(* CODESYS project fscontrollertoolbox_0.1.0.library
   Company: FisoThemes
   DocFormat: reStructuredText
   Description: A library for building and modelling control systems.
   Version: 0.1.0
   Placeholder: FsControllerToolbox
   Author: Goodwill Mzumala
   Title: FsControllerToolbox

Project tree, tasks and I/O mapping:
  libraries: FsCommon, * (FisoThemes); Tc2_Standard, * (Beckhoff Automation GmbH); Tc2_System, * (Beckhoff Automation GmbH); Tc3_Module, * (Beckhoff Automation GmbH); Tc2_Math, * (Beckhoff Automation GmbH)
  Analysis/
  Conditioning/
    DUTs/
      data type E_DeadbandMode
    function block FB_Deadband [ST]: FB_init, Maximum, Minimum, Mode, Reset, Run
    function block FB_Hysteresis [ST]: FB_init, LowerThreshold, Output, Reset, Run, UpperThreshold
  Control/
    DUTs/
      data type E_AntiWindupMethod
    function block FB_Differentiator [ST]: FB_init, Reset, Run, Td, Tv
    function block FB_Integrator [ST]: AntiWindupActive, AntiWindupMethod, FB_init, Maximum, Minimum, Reset, Run, Sync, Tn, TrackingTimeConstant
    function block FB_ProportionalGain [ST]: FB_init, Kp, Reset, Run
  Filter/
    function block FB_FirstOrderIIRFilter [ST]: Alpha, FB_init, Reset, Run
  Internal/
    program PLAYGROUND [ST]
  Project Information/
    function F_GetCompany [ST]
    function F_GetTitle [ST]
    function F_GetVersion [ST]
  Shared/
    ITFs/
      interface I_Component
      interface I_Resettable: Reset
      interface I_SiComponent: Input
      interface I_SisoComponent: Input, Output
      interface I_SoComponent: Output
    function block FB_SiComponent [ST]: Input
    function block FB_SisoComponent [ST]: Input, Output
    function block FB_SoComponent [ST]: Output
  Signals/
    DUTs/
      data type E_RampDirection
    ITFs/
      interface I_PeriodicSignal: Amplitude, Bias, Period, Phase
    function block FB_PeriodicSignal [ST]: Amplitude, Bias, Period, Phase
    function block FB_PWM [ST]: DutyCycle, FB_init, IsHigh, Reset, Run
    function block FB_Ramp [ST]: FB_init, Rate, Reset, Run, StartValue
    function block FB_SawtoothWave [ST]: Direction, FB_init, Reset, Run
    function block FB_SineWave [ST]: FB_init, Reset, Run
    function block FB_SquareWave [ST]: FB_init, Reset, Run
    function block FB_TriangleWave [ST]: FB_init, Reset, Run
  Simulation/
    function block FB_FirstOrderPlant [ST]: FB_init, Gain, Reset, Run, Tau
    function block FB_SecondOrderPlant [ST]: FB_init, Gain, Reset, Run, Wn, Zeta
  Transform/
  Version/
    global variables Global_Version
*)

// Conditioning/DUTs/E_DeadbandMode
(*
Specifies the behaviour of :itf:`FB_Deadband` when the input is within the band.
*)
{attribute 'qualified_only'}
{attribute 'strict'}
{attrubute 'to_string'}
TYPE E_DeadbandMode :
(
	Hold := 0, // Output holds its last value while the input is within the band.
	Zero := 1  // Output is set to zero while the input is within the band.
)BYTE;
END_TYPE

// Control/DUTs/E_AntiWindupMethod
(*
Specifies the anti-windup strategy used by :itf:`FB_Integrator`.
*)
{attribute 'qualified_only'}
{attribute 'strict'}
{attribute 'to_string'}
TYPE E_AntiWindupMethod :
(
	// Halts integration when the output is saturated.
	Clamping        := 0, 
	// Feeds back the saturation error to unwind the integrator gradually. 
	// Recommended for slow systems with significant lag
	BackCalculation := 1
)BYTE;
END_TYPE

// Signals/DUTs/E_RampDirection
(* Specifies the direction of a ramping signal. *)
{attribute 'qualified_only'}
{attribute 'strict'}
{attribute 'to_string'}
TYPE E_RampDirection :
(
	Rising   := 0, // Output increases over time.
	Falling  := 1  // Output decreases over time.
)BYTE;
END_TYPE

// Version/Global_Version
{attribute 'TcGenerated'}
{attribute 'no-analysis'}
{attribute 'linkalways'}
// This function has been automatically generated from the project information.
VAR_GLOBAL CONSTANT
	{attribute 'const_non_replaced'}
	stLibVersion_FsControllerToolbox : ST_LibVersion := (iMajor := 0, iMinor := 1, iBuild := 0, iRevision := 0, nFlags := 0, sVersion := '0.1.0');
END_VAR

// Conditioning/FB_Deadband
(*
Suppresses small input signals within a configurable band.

When the input falls within [:attr:`Minimum`, :attr:`Maximum`], the output
is either zeroed or held at its last value depending on :attr:`Mode`. Outside
the band the input passes through unchanged.

.. note::
   The block is ``FINAL`` and must be instantiated, not extended.
   Use ``FB_init`` to set :attr:`fMinimum`, :attr:`fMaximum`, and :attr:`eMode`
   at declaration time.
*)
{attribute 'no_assign'}
{attribute 'enable_dynamic_creation'}
{attribute 'no_explicit_call' := 'direct call for this function block is not allowed'}
FUNCTION_BLOCK FINAL FB_Deadband EXTENDS FB_SisoComponent
IMPLEMENTS FsCommon.I_Runnable, I_Resettable
VAR
	_fMinimum : LREAL; // Lower bound of the deadband. Clamped to <= Maximum.
	_fMaximum : LREAL; // Upper bound of the deadband. Clamped to >= Minimum.
	_eMode    : E_DeadbandMode; // Output behaviour when input is within the band.
END_VAR

METHOD FB_init : BOOL
VAR_INPUT
	bInitRetains : BOOL;  // if TRUE, the retain variables are initialized (warm start / cold start)
	bInCopyCode  : BOOL;  // if TRUE, the instance afterwards gets moved into the copy code (online change)
	fMaximum     : LREAL; // Upper bound of the deadband.
	fMinimum     : LREAL; // Lower bound of the deadband.
	eMode        : E_DeadbandMode; // Output behaviour when the input is within the band.
END_VAR
THIS^.Maximum  := fMaximum;
THIS^.Minimum  := fMinimum;
THIS^._eMode   := eMode;
END_METHOD

(*
Gets or sets the upper bound of the deadband.

Internally clamped to be greater than or equal to :attr:`Minimum`.
Set this before :attr:`Minimum` to ensure the guard applies correctly.
*)
PROPERTY Maximum : LREAL
GET
Maximum := THIS^._fMaximum;
END_GET
SET
THIS^._fMaximum := MAX(THIS^._fMinimum, Maximum);
END_SET
END_PROPERTY

(*
Gets or sets the lower bound of the deadband.

Internally clamped to be less than or equal to :attr:`Maximum`.
Set :attr:`Maximum` before this property to ensure the guard applies correctly.
*)
PROPERTY Minimum : LREAL
GET
Minimum := THIS^._fMinimum;
END_GET
SET
THIS^._fMinimum := MIN(THIS^._fMaximum, Minimum);
END_SET
END_PROPERTY

(*
Gets or sets the output behaviour when the input is within the band.

:attr:`~E_DeadbandMode.Zero` sets the output to zero. 
:attr:`~E_DeadbandMode.Hold` retains the last output value. 

Changes take effect on th next :meth:`Run` call.
*)
PROPERTY Mode : E_DeadbandMode
GET
Mode := THIS^._eMode;
END_GET
SET
THIS^._eMode := Mode;
END_SET
END_PROPERTY

(* 
Resets the output to a value consistent with the current mode. 

In :attr:`~E_DeadbandMode.Zero` mode the output is set to zero.
In :attr:`~E_DeadbandMode.Hold` mode the output is set to the current input.
*)
METHOD Reset
VAR_INPUT
END_VAR
CASE THIS^._eMode OF
	E_DeadbandMode.Hold:
		THIS^._fOutput := THIS^._fInput;
	E_DeadbandMode.Zero:
		THIS^._fOutput := 0;
END_CASE
END_METHOD

(* Applies the deadband to the current input. *)
METHOD Run
VAR_INPUT
END_VAR
THIS^._fMaximum := MAX(THIS^._fMinimum, THIS^._fMaximum);
THIS^._fMinimum := MIN(THIS^._fMinimum, THIS^._fMaximum);

IF THIS^._fInput >= THIS^._fMinimum AND THIS^._fInput <= THIS^._fMaximum THEN
    CASE THIS^._eMode OF
        E_DeadbandMode.Zero:
            THIS^._fOutput := 0;
        E_DeadbandMode.Hold:
            ; // Output retains its last value.
    END_CASE
ELSE
    THIS^._fOutput := THIS^._fInput;
END_IF
END_METHOD

END_FUNCTION_BLOCK

// Shared/FB_SisoComponent
(*
Abstract function block providing :attr:`Input` and :attr:`Output` properties
for single-input single-output controller toolbox components.

.. NOTE::
   Direct calls to this function block are not permitted (``no_explicit_call``).
*)
{attribute 'no_explicit_call' := 'direct call for this function block is not allowed'}
FUNCTION_BLOCK ABSTRACT FB_SisoComponent
IMPLEMENTS I_SisoComponent, I_SiComponent, I_SoComponent
VAR
	_fInput 	: LREAL;
	_fOutput 	: LREAL;
END_VAR

(* Gets or sets the input to the component.*)
PROPERTY Input : LREAL
GET
Input := THIS^._fInput;
END_GET
SET
THIS^._fInput := Input;
END_SET
END_PROPERTY

(* Gets the output produced by the component.*)
PROPERTY Output : LREAL
GET
Output := THIS^._fOutput;
END_GET
END_PROPERTY

END_FUNCTION_BLOCK

// Shared/ITFs/I_SisoComponent
(*
Interface for single-input single-output controller toolbox components.

Implementors expose a writable :attr:`Input` and a read-only :attr:`Output`,
both as ``LREAL``.
*)
INTERFACE I_SisoComponent EXTENDS I_Component

// Gets or sets the input to the component.
PROPERTY Input : LREAL
GET
END_GET
SET
END_SET
END_PROPERTY

// Gets the output produced by the component.
PROPERTY Output : LREAL
GET
END_GET
END_PROPERTY

END_INTERFACE

// Shared/ITFs/I_Component
(*
Base interface for all FsControllerToolbox components.

Extends ``__SYSTEM.IQueryInterface`` to allow runtime type checking via
``__QUERYINTERFACE``.
*)
INTERFACE I_Component EXTENDS __SYSTEM.IQueryInterface

END_INTERFACE

// Shared/ITFs/I_SiComponent
(*
Interface for single-input controller toolbox components.

Implementors expose a write-only :attr:`Input` property. For components that
also produce an output signal, use :itf:`I_SisoComponent` instead.
*)
INTERFACE I_SiComponent

// Gets or sets the input to the component.
PROPERTY Input : LREAL
GET
END_GET
SET
END_SET
END_PROPERTY

END_INTERFACE

// Shared/ITFs/I_SoComponent
(*
Interface for single-output controller toolbox components.

Implementors expose a read-only :attr:`Output` property. For components that
also accept an input signal, use :itf:`I_SisoComponent` instead.
*)
INTERFACE I_SoComponent EXTENDS I_Component

// Gets the output produced by the component.
PROPERTY Output : LREAL
GET
END_GET
END_PROPERTY

END_INTERFACE

// Shared/ITFs/I_Resettable
(*
Interface for components that can be returned to a known initial state.

Implementors must define :meth:`Reset` to clear any internal state, such as
accumulators, filter history, or elapsed time, and restore the output to its
initial condition.
*)
INTERFACE I_Resettable EXTENDS __SYSTEM.IQueryInterface

(* Clears internal state and restores the component to its initial condition. *)
METHOD Reset
VAR_INPUT
END_VAR
END_METHOD

END_INTERFACE

// Conditioning/FB_Hysteresis
(*
Implements a hysteresis controller with two thresholds and latching behaviour.

The output switches low when the input rises above :attr:`UpperThreshold` and
switches high when the input falls below :attr:`LowerThreshold`. Between the
two thresholds the output latches at its current state.

This convention suits heating applications, the output drives a heater that
turns on when the process falls below the lower threshold and off when it
exceeds the upper threshold.

.. note::
   The block is ``FINAL`` and must be instantiated, not extended.
   Use ``FB_init`` to set :attr:`fUpperThreshold` and :attr:`fLowerThreshold`
   at declaration time.
*)
{attribute 'no_assign'}
{attribute 'enable_dynamic_creation'}
{attribute 'no_explicit_call' := 'direct call for this function block is not allowed'}
FUNCTION_BLOCK FINAL FB_Hysteresis EXTENDS FB_SiComponent
IMPLEMENTS FsCommon.I_Runnable, I_Resettable
VAR
	_fUpperThreshold : LREAL; // Input level above which the output switches low.
	_fLowerThreshold : LREAL; // Input level below which the output switches high.
	_bOutput         : BOOL;  // Current output state.
END_VAR

METHOD FB_init : BOOL
VAR_INPUT
	bInitRetains 	 : BOOL; // if TRUE, the retain variables are initialized (warm start / cold start)
	bInCopyCode 	 : BOOL;  // if TRUE, the instance afterwards gets moved into the copy code (online change)
	fUpperThreshold  : LREAL; // Input level above which the output switches low.
	fLowerThreshold  : LREAL; // Input level below which the output switches high.
END_VAR
THIS^._fUpperThreshold := fUpperThreshold;
THIS^._fLowerThreshold := fLowerThreshold;
END_METHOD

(*
Gets or sets the lower threshold.

When the input falls below this value the output switches high. Must be less
than :attr:`UpperThreshold` for correct operation.
*)
PROPERTY LowerThreshold : LREAL
GET
LowerThreshold := THIS^._fLowerThreshold;
END_GET
SET
THIS^._fLowerThreshold := LowerThreshold;
END_SET
END_PROPERTY

(*
Gets the current output state. 

TRUE when the process is below :attr:`LowerThreshold`.
FALSE when above :attr:`UpperThreshold`.
*)
PROPERTY Output : BOOL
GET
Output := THIS^._bOutput;
END_GET
END_PROPERTY

(*
Evaluates the current input against the thresholds and sets the output immediately,
rather than waiting for the input to cross a threshold.

If the input is above :attr:`UpperThreshold` the output is set low. If below
:attr:`LowerThreshold` the output is set high. If between the two thresholds
the output defaults to low as a safe state.
*)
METHOD Reset
VAR_INPUT
END_VAR
THIS^._bOutput := THIS^._fInput < THIS^._fLowerThreshold;
END_METHOD

(* Evaluates the input against the thresholds and updates the output. *)
METHOD Run
VAR_INPUT
END_VAR
IF THIS^._fInput > THIS^._fUpperThreshold THEN
	THIS^._bOutput := FALSE;
ELSIF THIS^._fInput < THIS^._fLowerThreshold THEN
	THIS^._bOutput := TRUE;
END_IF
END_METHOD

(*
Gets or sets the upper threshold.

When the input rises above this value the output switches low. Must be greater
than :attr:`LowerThreshold` for correct operation.
*)
PROPERTY UpperThreshold : LREAL
GET
UpperThreshold := THIS^._fUpperThreshold;
END_GET
SET
THIS^._fUpperThreshold := UpperThreshold;
END_SET
END_PROPERTY

END_FUNCTION_BLOCK

// Shared/FB_SiComponent
(*
Abstract function block providing an :attr:`Input` property for single-input
controller toolbox components.

Concrete implementations read from ``_fInput`` to consume the signal written
by the caller.

.. note::
   Direct calls to this function block are not permitted (``no_explicit_call``).
   Extend it and call the derived block instead.
*)
{attribute 'no_explicit_call' := 'direct call for this function block is not allowed'}
FUNCTION_BLOCK ABSTRACT FB_SiComponent
IMPLEMENTS I_SiComponent
VAR
    _fInput : LREAL;
END_VAR

(* Gets or sets the input to the component.*)
PROPERTY Input : LREAL
GET
Input := THIS^._fInput;
END_GET
SET
THIS^._fInput := Input;
END_SET
END_PROPERTY

END_FUNCTION_BLOCK

// Control/FB_Differentiator
(*
Differentiates the input signal with an optional first-order damping filter.

The transfer function is:

.. math::

   D(s) = \frac{T_v \cdot s}{T_d \cdot s + 1}

where :math:`T_v` is :attr:`Tv` and :math:`T_d` is :attr:`Td`. The filter is
discretised using the Tustin (bilinear) method.

Setting :attr:`Tv` to ``LTIME#0`` disables the derivative term entirely.
Setting :attr:`Td` to ``LTIME#0`` removes the damping filter, giving a pure
derivative. This is not recommended in practice due to noise sensitivity.

.. note::
   If derivative kick on setpoint steps is undesirable, pass the negated
   process variable as :attr:`Input` rather than the full error. The integrator
   should still receive the full error signal.

   The block is ``FINAL`` and must be instantiated, not extended.
   Use ``FB_init`` to set :attr:`tTv` and :attr:`tTd` at declaration time.
*)
{attribute 'no_assign'}
{attribute 'enable_dynamic_creation'}
{attribute 'no_explicit_call' := 'direct call for this function block is not allowed'}
FUNCTION_BLOCK FINAL FB_Differentiator EXTENDS FB_SisoComponent
IMPLEMENTS FsCommon.I_Runnable, I_Resettable
VAR
	_tTv          : LTIME; // Rate time (Tv). Determines derivative action strength.
	_tTd          : LTIME; // Damping time (Td). Filters the derivative signal to reduce noise sensitivity.
	_fPrevInput   : LREAL; // Input from the previous cycle.
	_fFilterState : LREAL; // Internal state of the damping filter.
END_VAR

METHOD FB_init : BOOL
VAR_INPUT
	bInitRetains : BOOL; // if TRUE, the retain variables are initialized (warm start / cold start)
	bInCopyCode  : BOOL;  // if TRUE, the instance afterwards gets moved into the copy code (online change)
	tTv          : LTIME; // Rate time. T#0S disables the derivative term entirely.
	tTd          : LTIME; // Damping time. LTIME#0 means no filtering (pure derivative).
END_VAR
THIS^._tTv := tTv;
THIS^._tTd := tTd;
END_METHOD

(*
Clears the filter state and output. 
Sets the previous input to the current input to avoid a spike on the next :meth:`Run` call. 
*)
METHOD Reset
VAR_INPUT
END_VAR
THIS^._fFilterState := 0;
THIS^._fPrevInput   := THIS^._fInput;
THIS^._fOutput      := 0;
END_METHOD

(*
Advances the differentiator by one time step.

On the first call the cycle time is measured, the filter state is initialised,
and the method returns early without producing an output. This prevents a spike
caused by an uninitialised previous input.

.. note::
   Must be called once per cycle on a single PLC task. If :attr:`Tv` is
   ``LTIME#0`` the output is held at zero.
*)
METHOD Run
VAR_INST
	{attribute 'hide'}
	bInit       : BOOL := TRUE;
	{attribute 'hide'}
	fT          : LREAL;
	{attribute 'hide'}
	fbTaskCycle : FsCommon.FB_PlcTaskCycleChangeDetector(0);
END_VAR
VAR
	fTv            : LREAL;
	fTd            : LREAL;
	fDen           : LREAL;
	fAlpha         : LREAL;
	fRawDerivative : LREAL;
END_VAR
IF bInit THEN
	fT := TO_LREAL(FsCommon.F_GetCurrentTaskCycleTime()) / TO_LREAL(LTIME#1S);
	RETURN(bInit := fT <= 0);
	fbTaskCycle.TaskIndex := FsCommon.F_GetCurrentTaskIndex();
	THIS^._fPrevInput     := THIS^._fInput;
	THIS^._fFilterState   := 0;
	RETURN;
END_IF

RETURN(NOT fbTaskCycle.HasChanged);

IF THIS^._tTv = LTIME#0S THEN
	THIS^._fOutput    := 0;
	THIS^._fPrevInput := THIS^._fInput;
	RETURN;
END_IF

fTv := TO_LREAL(THIS^._tTv) / TO_LREAL(LTIME#1S);
fTd := TO_LREAL(THIS^._tTd) / TO_LREAL(LTIME#1S);

fRawDerivative := fTv * (THIS^._fInput - THIS^._fPrevInput) / fT;

IF THIS^._tTd = LTIME#0S THEN
	THIS^._fOutput := fRawDerivative;
ELSE
	fDen                := fTd + fT / 2.0;
	fAlpha              := (fTd - fT / 2.0) / fDen;
	THIS^._fFilterState := fAlpha * THIS^._fFilterState + (1.0 - fAlpha) * fRawDerivative;
	THIS^._fOutput      := THIS^._fFilterState;
END_IF

THIS^._fPrevInput := THIS^._fInput;
END_METHOD

(*
Gets or sets the damping time (Td).

This filters the derivative signal to reduce sensitivity to noise. A longer
value gives more filtering but reduces derivative effectiveness. Setting it
to ``LTIME#0`` removes the filter entirely, giving a pure derivative (not
recommended in practice due to noise sensitivity).
*)
PROPERTY Td : LTIME
GET
Td := THIS^._tTd;
END_GET
SET
THIS^._tTd := Td;
END_SET
END_PROPERTY

(*
Gets or sets the rate time (Tv).

This controls how strongly the block reacts to changes in the input. A longer
value increases derivative action. Setting it to ``LTIME#0`` disables the
derivative term entirely, holding the output at zero.
*)
PROPERTY Tv : LTIME
GET
Tv := THIS^._tTv;
END_GET
SET
THIS^._tTv := Tv;
END_SET
END_PROPERTY

END_FUNCTION_BLOCK

// Control/FB_Integrator
(*
Integrates the input error signal over time.

The output accumulates the input scaled by the integral gain :math:`K_i = 1 / T_n`,
and is clamped to [:attr:`Minimum`, :attr:`Maximum`] on every cycle. Two anti-windup
strategies are available via :attr:`AntiWindupMethod`.

Setting :attr:`Tn` to ``LTIME#0`` disables integration, holding the output at
its current integrator state.

.. note::
   Set :attr:`Maximum` before :attr:`Minimum` to ensure the clamp is applied
   correctly. Setting :attr:`Minimum` first may cause it to be clamped against
   an uninitialised :attr:`Maximum`.

   The block is ``FINAL`` and must be instantiated, not extended.
   Use ``FB_init`` to set :attr:`tTn`, :attr:`fMaximum`, :attr:`fMinimum`,
   :attr:`eAntiWindupMethod`, and :attr:`tTrackingTimeConstant` at declaration time.
*)
{attribute 'no_assign'}
{attribute 'enable_dynamic_creation'}
{attribute 'no_explicit_call' := 'direct call for this function block is not allowed'}
FUNCTION_BLOCK FINAL FB_Integrator EXTENDS FB_SisoComponent
IMPLEMENTS FsCommon.I_Runnable, I_Resettable
VAR
	_tTn                   : LTIME; // Integral action time (Tn).
	_fMaximum              : LREAL :=  FsCommon.GVL_TypeValueLimits.LREAL_MAX; // Upper output clamp.
	_fMinimum              : LREAL :=  FsCommon.GVL_TypeValueLimits.LREAL_MIN; // Lower output clamp.
	_eAntiWindupMethod     : E_AntiWindupMethod; // Anti-windup strategy.
	_tTrackingTimeConstant : LTIME; // Tracking time constant (Tt) for back-calculation anti-windup.
	_fIntegratorState      : LREAL; // Internal integrator accumulator.
	_bAntiWindupActive     : BOOL;  // TRUE when the output is saturated and anti-windup is limiting integration.
	_bSync                 : BOOL;  // Triggers a bumpless transfer on the next Run call.
	_fSync                 : LREAL; // Target integrator state for bumpless transfer.
END_VAR

(* Gets whether the output is currently saturated and anti-windup is actively limiting integration. *)
PROPERTY AntiWindupActive : BOOL
GET
AntiWindupActive := THIS^._bAntiWindupActive;
END_GET
END_PROPERTY

(*
Gets or sets the anti-windup strategy.

:attr:`~E_AntiWindupMethod.Clamping` halts integration when the output is
saturated. :attr:`~E_AntiWindupMethod.BackCalculation` feeds the saturation
error back into the integrator gradually, which is better suited to slow
systems with significant lag such as thermal processes.
*)
PROPERTY AntiWindupMethod : E_AntiWindupMethod
GET
AntiWindupMethod := THIS^._eAntiWindupMethod;
END_GET
SET
THIS^._eAntiWindupMethod := AntiWindupMethod;
END_SET
END_PROPERTY

METHOD FB_init : BOOL
VAR_INPUT
	bInitRetains 		  : BOOL;  // if TRUE, the retain variables are initialized (warm start / cold start)
	bInCopyCode 		  : BOOL;  // if TRUE, the instance afterwards gets moved into the copy code (online change)
	tTn                   : LTIME; // Integral action time. LTIME#0 disables integration.
	fMaximum              : LREAL; // Upper output clamp.
	fMinimum              : LREAL; // Lower output clamp.
	eAntiWindupMethod     : E_AntiWindupMethod; // Anti-windup strategy.
	tTrackingTimeConstant : LTIME; // Tracking time constant for back-calculation anti-windup.
END_VAR
THIS^._tTn                   := tTn;
THIS^.Maximum                := fMaximum;
THIS^.Minimum                := fMinimum;
THIS^._eAntiWindupMethod     := eAntiWindupMethod;
THIS^._tTrackingTimeConstant := tTrackingTimeConstant;
END_METHOD

(*
Gets or sets the upper output clamp.

The output is clamped to this value on every cycle. Internally clamped to be
greater than or equal to :attr:`Minimum`. Set this before :attr:`Minimum` to
ensure the guard applies correctly.
*)
PROPERTY Maximum : LREAL
GET
Maximum := THIS^._fMaximum;
END_GET
SET
THIS^._fMaximum := MAX(THIS^._fMinimum, Maximum);
END_SET
END_PROPERTY

(*
Gets or sets the lower output clamp.

The output is clamped to this value on every cycle. Internally clamped to be
less than or equal to :attr:`Maximum`. Set :attr:`Maximum` before this property
to ensure the guard applies correctly.
*)
PROPERTY Minimum : LREAL
GET
Minimum := THIS^._fMinimum;
END_GET
SET
THIS^._fMinimum := MIN(THIS^._fMaximum, Minimum);
END_SET
END_PROPERTY

(* Clears the integrator state, output, and anti-windup flag. *)
METHOD Reset
VAR_INPUT
END_VAR
THIS^._fIntegratorState  := 0;
THIS^._fOutput           := 0;
THIS^._bAntiWindupActive := FALSE;
END_METHOD

(*
Advances the integrator by one time step.

.. note::
   Must be called once per cycle on a single PLC task. If :attr:`Tn` is
   ``LTIME#0`` the output is held at the current integrator state without
   further integration.
*)
METHOD Run
VAR_INST
	{attribute 'hide'}
	bInit       : BOOL := TRUE;
	{attribute 'hide'}
	fT          : LREAL;
	{attribute 'hide'}
	fbTaskCycle : FsCommon.FB_PlcTaskCycleChangeDetector(0);
END_VAR
VAR
	fKi                   : LREAL;
	fTt                   : LREAL;
	fWindupBack           : LREAL;
	fUnsat                : LREAL;
	fSaturated            : LREAL;
END_VAR
IF bInit THEN
	fT := TO_LREAL(FsCommon.F_GetCurrentTaskCycleTime()) / TO_LREAL(LTIME#1S);
	RETURN(bInit := fT <= 0);
	fbTaskCycle.TaskIndex := FsCommon.F_GetCurrentTaskIndex();
END_IF

THIS^._fMaximum := MAX(THIS^._fMinimum, THIS^._fMaximum);
THIS^._fMinimum := MIN(THIS^._fMinimum, THIS^._fMaximum);

RETURN(NOT fbTaskCycle.HasChanged);

// Bumpless transfer, force integrator state before anything else.
IF FsCommon.F_ResetOnTrue(THIS^._bSync) THEN
	THIS^._fIntegratorState := LIMIT(THIS^._fMinimum, THIS^._fSync, THIS^._fMaximum);
END_IF

IF THIS^._tTn = LTIME#0S THEN
	THIS^._fOutput := THIS^._fIntegratorState;
	RETURN;
END_IF

fKi := 1.0 / (TO_LREAL(THIS^._tTn) / TO_LREAL(LTIME#1S));

CASE THIS^._eAntiWindupMethod OF
	E_AntiWindupMethod.Clamping:
		IF NOT THIS^._bAntiWindupActive OR
		   (THIS^._fOutput >= THIS^._fMaximum AND THIS^._fInput < 0) OR
		   (THIS^._fOutput <= THIS^._fMinimum AND THIS^._fInput > 0) THEN
			THIS^._fIntegratorState :=
				THIS^._fIntegratorState + fKi * THIS^._fInput * fT;
		END_IF

	E_AntiWindupMethod.BackCalculation:
		fTt := TO_LREAL(THIS^._tTrackingTimeConstant) / TO_LREAL(LTIME#1S);
		fWindupBack := SEL(
			fTt > 0,
			0.0,
			(THIS^._fOutput - THIS^._fIntegratorState) / fTt);
		THIS^._fIntegratorState :=
			THIS^._fIntegratorState + (fKi * THIS^._fInput + fWindupBack) * fT;
END_CASE

fUnsat                   := THIS^._fIntegratorState;
fSaturated               := LIMIT(THIS^._fMinimum, fUnsat, THIS^._fMaximum);
THIS^._bAntiWindupActive := fSaturated <> fUnsat;
THIS^._fOutput           := fSaturated;
END_METHOD

(*
Forces the integrator state to a given value on the next :meth:`Run` call.

The value is clamped to [:attr:`Minimum`, :attr:`Maximum`] before being applied.
Use this for bumpless transfer when switching from manual to automatic mode,
to prevent a sudden jump in output.
*)
METHOD Sync
VAR_INPUT
	// Target integrator state.
	fValue : LREAL; 
END_VAR
THIS^._bSync := TRUE;
THIS^._fSync := LIMIT(THIS^._fMinimum, fValue, THIS^._fMaximum);
END_METHOD

(*
Gets or sets the integral action time (Tn).

This controls how aggressively the integrator responds to sustained error.
A shorter value increases integral action. Setting it to ``LTIME#0`` disables
integration entirely, holding the output at the current integrator state.
*)
PROPERTY Tn : LTIME
GET
Tn := THIS^._tTn;
END_GET
SET
THIS^._tTn := Tn;
END_SET
END_PROPERTY

(*
Gets or sets the tracking time constant (Tt) for back-calculation anti-windup.

This controls how quickly the integrator unwinds after saturation. A typical
starting value is ``SQRT(Tn * Td)``. Setting it to ``LTIME#0`` disables the
back-calculation correction. Ignored when :attr:`AntiWindupMethod` is
:attr:`~E_AntiWindupMethod.Clamping`.
*)
PROPERTY TrackingTimeConstant : LTIME
GET
TrackingTimeConstant := THIS^._tTrackingTimeConstant;
END_GET
SET
THIS^._tTrackingTimeConstant := TrackingTimeConstant;
END_SET
END_PROPERTY

END_FUNCTION_BLOCK

// Control/FB_ProportionalGain
(*
Applies a proportional gain to the input error signal.

The output is computed as:

.. math::

   y = K_p \cdot e

where :math:`K_p` is :attr:`Kp` and :math:`e` is the error signal set via :attr:`Input`.

.. note::
   The block is ``FINAL`` and must be instantiated, not extended.
   Use ``FB_init`` to set :attr:`fKp` at declaration time.
*)
{attribute 'no_assign'}
{attribute 'enable_dynamic_creation'}
{attribute 'no_explicit_call' := 'direct call for this function block is not allowed'}
FUNCTION_BLOCK FINAL FB_ProportionalGain EXTENDS FB_SisoComponent
IMPLEMENTS FsCommon.I_Runnable, I_Resettable
VAR
	_fKp : LREAL; // Proportional gain.
END_VAR

METHOD FB_init : BOOL
VAR_INPUT
	bInitRetains : BOOL; // if TRUE, the retain variables are initialized (warm start / cold start)
	bInCopyCode  : BOOL;  // if TRUE, the instance afterwards gets moved into the copy code (online change)
	fKp          : LREAL; // Proportional gain.
END_VAR
THIS^._fKp := fKp;
END_METHOD

(*
Gets or sets the proportional gain.

A higher value produces a stronger response to error but may cause overshoot.
A lower value produces a more gradual response. A value of 0 disables the
proportional term entirely.
*)
PROPERTY Kp : LREAL
GET
Kp := THIS^._fKp;
END_GET
SET
THIS^._fKp := Kp;
END_SET
END_PROPERTY

(* Sets the output to zero. Takes effect until the next :meth:`Run` call. *)
METHOD Reset
VAR_INPUT
END_VAR
THIS^._fOutput := 0;
END_METHOD

(*
Computes the proportional output for the current cycle.

.. note::
   Must be called once per cycle on a single PLC task.
*)
METHOD Run
VAR_INPUT
END_VAR
THIS^._fOutput := THIS^._fKp * THIS^._fInput;
END_METHOD

END_FUNCTION_BLOCK

// Filter/FB_FirstOrderIIRFilter
(*
Applies an exponential moving average (EMA) to the input signal.

On the first call the output is set to the current input. On subsequent calls:

.. math::

   y[k] = \alpha \cdot u[k] + (1 - \alpha) \cdot y[k-1]

where :math:`\alpha` is :attr:`Alpha`. A value of 0 passes the input through
unchanged. A value of 1 holds the output at the first input value.

.. note::
   The block is ``FINAL`` and must be instantiated, not extended.
   Use ``FB_init`` to set :attr:`fAlpha` at declaration time.
*)
{attribute 'no_assign'}
{attribute 'enable_dynamic_creation'}
{attribute 'no_explicit_call' := 'direct call for this function block is not allowed'}
FUNCTION_BLOCK FINAL FB_FirstOrderIIRFilter EXTENDS FB_SisoComponent
IMPLEMENTS FsCommon.I_Runnable, I_Resettable
VAR
	_fAlpha : LREAL; // Smoothing factor. Clamped to 0..1.
END_VAR

(*
Gets or sets the smoothing factor.

Controls the balance between the current input and the previous output.
A value closer to 0 produces a smoother, slower-responding output. A value
closer to 1 tracks the input more closely with less smoothing.
Values outside 0..1 are clamped.
*)
PROPERTY Alpha : LREAL
GET
Alpha := THIS^._fAlpha;
END_GET
SET
THIS^._fAlpha := LIMIT(0, Alpha, 1);
END_SET
END_PROPERTY

METHOD FB_init : BOOL
VAR_INPUT
	bInitRetains : BOOL; // if TRUE, the retain variables are initialized (warm start / cold start)
	bInCopyCode  : BOOL;  // if TRUE, the instance afterwards gets moved into the copy code (online change)
	fAlpha       : LREAL; // Smoothing factor. Clamped to 0..1.
END_VAR
THIS^._fAlpha := LIMIT(0, fAlpha, 1);
END_METHOD

(*
Sets the output to zero. 
On the next :meth:`Run` call the output will reinitialise to the current input.
*)
METHOD Reset
VAR_INPUT
END_VAR
THIS^._fOutput := 0;
END_METHOD

(*
Advances the filter by one time step.

On the first call the output is initialised to the current input to avoid
a transient caused by a zero initial state. Subsequent calls apply the
exponential moving average.
*)
METHOD Run
VAR_INST
	{attribute 'hide'}
	bInit : BOOL := TRUE;
END_VAR
IF FsCommon.F_ResetOnTrue(bInit) THEN
	THIS^._fOutput := THIS^._fInput;
	RETURN;
END_IF

THIS^._fOutput := THIS^._fAlpha * THIS^._fInput + (1.0 - THIS^._fAlpha) * THIS^._fOutput;
END_METHOD

END_FUNCTION_BLOCK

// Internal/PLAYGROUND
PROGRAM INTERNAL PLAYGROUND
VAR
	fSetpoint : LREAL; 
	fError    : LREAL;
	fbPlant   : FB_FirstOrderPlant(fGain := 1.0, tTau := LTIME#5S);
	fbP       : FB_ProportionalGain(fKp := 2.0);
	fbI       : FB_Integrator(
					tTn 				  := LTIME#5S,
					fMaximum 			  := 100.0,
					fMinimum  			  := 0.0,
					eAntiWindupMethod 	  := E_AntiWindupMethod.BackCalculation,
					tTrackingTimeConstant := LTIME#2S200MS);
	fbD       : FB_Differentiator(tTv := LTIME#1S, tTd := LTIME#200MS);
END_VAR

fbP.Input := fError := fSetpoint - fbPlant.Output;
fbP.Run();
fbI.Input := fError;
fbI.Run();
fbD.Input := fError;
fbD.Run();

fbPlant.Input := fbP.Output + fbI.Output + fbD.Output;
fbPlant.Run();

END_PROGRAM

// Simulation/FB_FirstOrderPlant
(*
Simulates a first-order linear plant using Euler's backward (implicit) discretisation.

The continuous-time transfer function is:

.. math::

   G(s) = \frac{K}{\tau s + 1}

which discretises to:

.. math::

   y[k] = \frac{\tau \cdot y[k-1] + K \cdot \Delta t \cdot u[k]}{\tau + \Delta t}

where :math:`K` is :attr:`Gain`, :math:`\tau` is :attr:`Tau` in seconds, and
:math:`\Delta t` is the task cycle time, measured automatically on the first call.

.. note::
   The block is ``FINAL`` and must be instantiated, not extended.
   Use ``FB_init`` to set :attr:`fGain` and :attr:`fTau` at declaration time.
*)
{attribute 'enable_dynamic_creation'}
{attribute 'no_explicit_call' := 'direct call for this function block is not allowed'}
FUNCTION_BLOCK FINAL FB_FirstOrderPlant EXTENDS FB_SisoComponent
IMPLEMENTS FsCommon.I_Runnable, I_Resettable
VAR
	_fGain 	: LREAL; // Steady-state gain (K). Ratio of output to input once the plant has fully settled.
	_tTau 	: LTIME; // Time constant (τ). Time for the step response to reach 63.2% of its final value.
END_VAR

METHOD FB_init : BOOL
VAR_INPUT
	bInitRetains 	: BOOL;  // if TRUE, the retain variables are initialized (warm start / cold start)
	bInCopyCode 	: BOOL;  // if TRUE, the instance afterwards gets moved into the copy code (online change)
	fGain 			: LREAL; // Steady-state gain (K). Ratio of output to input once the plant has fully settled.
	tTau 			: LTIME; // Time constant (τ). Time for the step response to reach 63.2% of its final value.
END_VAR
THIS^._fGain := fGain;
THIS^._tTau  := tTau;
END_METHOD

(*
Gets or sets the steady-state gain.

This is the factor by which a constant input is scaled to produce the output once
the plant has fully settled. For example, a gain of 2 with a constant input of 5
will eventually produce an output of 10.
*)
PROPERTY Gain : LREAL
GET
Gain := THIS^._fGain;
END_GET
SET
THIS^._fGain := Gain;
END_SET
END_PROPERTY

(* Sets the output to zero, returning the plant to its initial state. *)
METHOD Reset
VAR_INPUT
END_VAR
THIS^._fOutput := 0;
END_METHOD

(*
Advances the plant by one time step.

.. note::
   Must be called once per cycle on a single PLC task. This is because on the 
   first call, the cycle time is measured and stored for use in all subsequent calls. 
 
   If the measured cycle time is zero the method returns early without updating 
   the output, guarding against a divide-by-zero.
*)
METHOD Run
VAR_INST
	{attribute 'hide'}
	bInit 	: BOOL := TRUE;
	{attribute 'hide'}
	fDt			: LREAL;
	{attribute 'hide'}
	fbTaskCycle :  FsCommon.FB_PlcTaskCycleChangeDetector(0);
END_VAR
VAR
	fTau 		: LREAL;
END_VAR
IF bInit THEN
	fDt := TO_LREAL(FsCommon.F_GetCurrentTaskCycleTime()) / TO_LREAL(LTIME#1S);
	RETURN(bInit := fDt <= 0);
	fbTaskCycle.TaskIndex := FsCommon.F_GetCurrentTaskIndex();
END_IF

RETURN(NOT fbTaskCycle.HasChanged);

fTau := TO_LREAL(THIS^._tTau) / TO_LREAL(LTIME#1S);

THIS^._fOutput := 
	(fTau * THIS^._fOutput + THIS^._fGain * fDt * THIS^._fInput) 
	/ 
	(fTau + fDt);
END_METHOD

(* 
Gets or sets the time constant (τ).

This controls how quickly the plant responds to a change in input. 
A larger value means a slower response. It is the time taken for the 
output to reach 63.2% of its final value after a step change in input.
*)
PROPERTY Tau : LTIME
GET
Tau := THIS^._tTau;
END_GET
SET
THIS^._tTau := Tau;
END_SET
END_PROPERTY

END_FUNCTION_BLOCK

// Project Information/F_GetCompany
// This function has been automatically generated from the project information.
{attribute 'signature_flag' := '1073741824'}
{attribute 'TcGenerated'}
{attribute 'no-analysis'}
FUNCTION F_GetCompany : WSTRING
VAR_INPUT
	
END_VAR

F_GetCompany := "FisoThemes";

END_FUNCTION

// Project Information/F_GetTitle
// This function has been automatically generated from the project information.
{attribute 'signature_flag' := '1073741824'}
{attribute 'TcGenerated'}
{attribute 'no-analysis'}
FUNCTION F_GetTitle : WSTRING
VAR_INPUT
	
END_VAR

F_GetTitle := "FsControllerToolbox";

END_FUNCTION

// Project Information/F_GetVersion
// This function has been automatically generated from the project information.
{attribute 'signature_flag' := '1073741824'}
{attribute 'TcGenerated'}
{attribute 'no-analysis'}
FUNCTION F_GetVersion : ST_LibVersion
VAR_INPUT
	
END_VAR

F_GetVersion.iMajor := 0;
F_GetVersion.iMinor := 1;
F_GetVersion.iBuild := 0;
F_GetVersion.iRevision := 0;
F_GetVersion.sVersion := '0.1.0';
F_GetVersion.nFlags := 0;

END_FUNCTION

// Shared/FB_SoComponent
(*
Abstract function block providing an :attr:`Output` property for single-output
controller toolbox components.

Concrete implementations must call this block cyclically and write their
result to ``_fOutput``.

.. note::
   Direct calls to this function block are not permitted (``no_explicit_call``).
   Extend it and call the derived block instead.
*)
{attribute 'no_explicit_call' := 'direct call for this function block is not allowed'}
FUNCTION_BLOCK ABSTRACT FB_SoComponent
IMPLEMENTS I_SoComponent
VAR
	_fOutput : LREAL;
END_VAR

(* Gets the output produced by the component.*)
PROPERTY Output : LREAL
GET
Output := THIS^._fOutput;
END_GET
END_PROPERTY

END_FUNCTION_BLOCK

// Signals/ITFs/I_PeriodicSignal
(*
Base interface for periodic signal generators.

Implementors produce a cyclic output defined by :attr:`Period`, :attr:`Amplitude`,
:attr:`Bias`, and :attr:`Phase`.
*)
INTERFACE I_PeriodicSignal EXTENDS I_SoComponent

(*
Gets or sets the amplitude. 

The output swings between ``Bias + Amplitude`` and ``Bias - Amplitude``.
*)
PROPERTY Amplitude : LREAL
GET
END_GET
SET
END_SET
END_PROPERTY

(*
Gets or sets the bias.

This is a fixed offset added to the output, shifting the wave up or down.
*)
PROPERTY Bias : LREAL
GET
END_GET
SET
END_SET
END_PROPERTY

(* 
Gets or sets the period. 

This is the time taken to complete one full cycle.
*)
PROPERTY Period : LTIME
GET
END_GET
SET
END_SET
END_PROPERTY

(*
Gets or sets the phase offset in radians.

This shifts the wave horizontally. Negative values shift in the opposite direction.
*)
PROPERTY Phase : LREAL
GET
END_GET
SET
END_SET
END_PROPERTY

END_INTERFACE

// Signals/FB_PeriodicSignal
(*
Abstract base block for periodic signal generators.

Provides :attr:`Period`, :attr:`Amplitude`, :attr:`Bias`, and :attr:`Phase`
as shared properties for all periodic signal generators. Derived blocks can
implement :meth:`Run` and :meth:`Reset` to produce their specific waveform.

.. note::
   Direct calls to this function block are not permitted (``no_explicit_call``).
   Extend it and call the derived block instead.
*)
{attribute 'enable_dynamic_creation'}
{attribute 'no_explicit_call' := 'direct call for this function block is not allowed'}
FUNCTION_BLOCK ABSTRACT FB_PeriodicSignal EXTENDS FB_SoComponent
IMPLEMENTS I_PeriodicSignal
VAR
	_tPeriod    : LTIME; // Duration of one full cycle. Must be greater than zero.
	_fAmplitude : LREAL; // Scales the raw wave. Output swings between Bias ± Amplitude.
	_fBias      : LREAL; // Shifts the output vertically.
	_fPhase     : LREAL; // Phase offset in radians. Shifts the wave horizontally.
END_VAR

(*
Gets or sets the amplitude. 

The output swings between ``Bias + Amplitude`` and ``Bias - Amplitude``.
*)
PROPERTY Amplitude : LREAL
GET
Amplitude := THIS^._fAmplitude;
END_GET
SET
THIS^._fAmplitude := Amplitude;
END_SET
END_PROPERTY

(*
Gets or sets the bias.

This is a fixed offset added to the output, shifting the wave up or down.
*)
PROPERTY Bias : LREAL
GET
Bias := THIS^._fBias;
END_GET
SET
THIS^._fBias := Bias;
END_SET
END_PROPERTY

(* 
Gets or sets the period. 

This is the time taken to complete one full cycle.
*)
PROPERTY Period : LTIME
GET
Period := THIS^._tPeriod;
END_GET
SET
THIS^._tPeriod := Period;
END_SET
END_PROPERTY

(*
Gets or sets the phase offset in radians.

This shifts the wave horizontally. Negative values shift in the opposite direction.
*)
PROPERTY Phase : LREAL
GET
Phase := THIS^._fPhase;
END_GET
SET
THIS^._fPhase := Phase;
END_SET
END_PROPERTY

END_FUNCTION_BLOCK

// Signals/FB_PWM
(*
Generates a pulse-width modulated (PWM) signal.

The output switches between ``Amplitude`` and ``0`` at a fixed :attr:`Period`.
:attr:`DutyCycle` controls the proportion of the period the output is high,
as a value between -1 and 1.

For example, a duty cycle of 0.3 produces a high output for 30% of the period
and a low output for the remaining 70%. A duty cycle of -0.3 inverts this,
producing a low output for 30% and a high output for 70%.

A duty cycle of 0 keeps the output permanently low. A duty cycle of ±1 keeps
it permanently high.

:attr:`Phase` shifts the wave horizontally in radians. Negative values shift
in the opposite direction.
:attr:`Bias` shifts the output vertically.

.. note::
   The block is ``FINAL`` and must be instantiated, not extended.
   Use ``FB_init`` to set :attr:`tPeriod`, :attr:`fAmplitude`, :attr:`fBias`,
   and :attr:`fDutyCycle` at declaration time.
*)
{attribute 'enable_dynamic_creation'}
{attribute 'no_explicit_call' := 'direct call for this function block is not allowed'}
FUNCTION_BLOCK FINAL FB_PWM EXTENDS FB_PeriodicSignal
IMPLEMENTS FsCommon.I_Runnable, I_Resettable
VAR
	_fDutyCycle : LREAL; // Proportion of the period the output is high. Clamped to -1..1. Negative values invert the wave.
	_bIsHigh    : BOOL;  // TRUE when the output is in its high state, regardless of amplitude, bias, or phase.
	{attribute 'hide'}
	_tTime      : LTIME;
END_VAR

(*
Gets or sets the duty cycle as a value between -1 and 1.

This controls the proportion of the period the output is high. A value of 0.3
keeps the output high for 30% of the period. A negative value inverts the wave —
-0.3 keeps the output low for 30% and high for the remaining 70%. Values outside
-1..1 are clamped. Changes take effect immediately.
*)
PROPERTY DutyCycle : LREAL
GET
DutyCycle := THIS^._fDutyCycle;
END_GET
SET
THIS^._fDutyCycle := LIMIT(-1, DutyCycle, 1);
END_SET
END_PROPERTY

METHOD FB_init : BOOL
VAR_INPUT
	bInitRetains : BOOL; // if TRUE, the retain variables are initialized (warm start / cold start)
	bInCopyCode : BOOL;  // if TRUE, the instance afterwards gets moved into the copy code (online change)
	tPeriod      : LTIME; // Duration of one full cycle.
	fAmplitude   : LREAL; // High-state output level. Low state is always 0.
	fBias        : LREAL; // Shifts the output vertically.
	fDutyCycle   : LREAL; // Proportion of the period the output is high. Clamped to -1..1.
END_VAR
THIS^._tPeriod    := tPeriod;
THIS^._fAmplitude := fAmplitude;
THIS^._fBias      := fBias;
THIS^._fDutyCycle := LIMIT(-1.0, fDutyCycle, 1.0);
END_METHOD

(*
Gets whether the output is currently in its high state.

TRUE regardless of the values of :attr:`Amplitude`, :attr:`Bias`, or :attr:`Phase`.
*)
PROPERTY IsHigh  : BOOL
GET
IsHigh := THIS^._bIsHigh;
END_GET
END_PROPERTY

(* 
Restarts the wave from the beginning by resetting the accumulated time to zero.
The duty cycle, phase, amplitude, and bias are unaffected.
*)
METHOD Reset
VAR_INPUT
END_VAR
THIS^._tTime  := LTIME#0S;
THIS^._bIsHigh := FALSE;
END_METHOD

(*
Advances the PWM signal by one time step.

.. note::
   Must be called once per cycle on a single PLC task. If the measured cycle
   time is zero or :attr:`Period` is zero, the method returns early without
   updating the output.
*)
METHOD Run
VAR_INST
	{attribute 'hide'}
	bInit       : BOOL := TRUE;
	{attribute 'hide'}
	fT          : LREAL;
	{attribute 'hide'}
	fbTaskCycle : FsCommon.FB_PlcTaskCycleChangeDetector(0);
END_VAR
VAR
	fPeriod    : LREAL;
	fPhaseTime : LREAL;
	fCyclePos  : LREAL;
	fDuty      : LREAL;
END_VAR
IF bInit THEN
	fT := TO_LREAL(FsCommon.F_GetCurrentTaskCycleTime()) / TO_LREAL(LTIME#1S);
	RETURN(bInit := fT <= 0);
	fbTaskCycle.TaskIndex := FsCommon.F_GetCurrentTaskIndex();
END_IF

RETURN(THIS^._tPeriod <= LTIME#0S OR NOT fbTaskCycle.HasChanged);

THIS^._tTime := THIS^._tTime + TO_LTIME(LREAL_TO_ULINT(fT * 1.0E9));

fPeriod    := TO_LREAL(THIS^._tPeriod) / TO_LREAL(LTIME#1S);
fPhaseTime := TO_LREAL(THIS^._tTime) / TO_LREAL(LTIME#1S) + (THIS^._fPhase / (2.0 * Tc2_System.PI)) * fPeriod;
fCyclePos  := Tc2_Math.LMOD(fPhaseTime, fPeriod) / fPeriod;

THIS^._fDutyCycle := LIMIT(-1, THIS^._fDutyCycle, 1);

fDuty := ABS(THIS^._fDutyCycle);

IF THIS^._fDutyCycle >= 0.0 THEN
	THIS^._bIsHigh := fCyclePos < fDuty;
ELSE
	THIS^._bIsHigh := fCyclePos >= (1.0 - fDuty);
END_IF

IF THIS^._bIsHigh THEN
	THIS^._fOutput := THIS^._fAmplitude + THIS^._fBias;
ELSE
	THIS^._fOutput := THIS^._fBias;
END_IF
END_METHOD

END_FUNCTION_BLOCK

// Signals/FB_Ramp
(*
Generates a ramp signal that rises or falls at a fixed rate indefinitely.

The output starts at :attr:`StartValue` and advances at :attr:`Rate` units per second.
A positive rate produces a rising ramp, a negative rate a falling ramp.
Changing :attr:`Rate` mid-run takes effect immediately.

Calling :meth:`Reset` returns the output to :attr:`StartValue`.

.. note::
   The block is ``FINAL`` and must be instantiated, not extended.
   Use ``FB_init`` to set :attr:`fStartValue` and :attr:`fRate` at declaration time.
*)
{attribute 'enable_dynamic_creation'}
{attribute 'no_explicit_call' := 'direct call for this function block is not allowed'}
FUNCTION_BLOCK FINAL FB_Ramp EXTENDS FB_SoComponent
IMPLEMENTS FsCommon.I_Runnable, I_Resettable
VAR
	_fStartValue : LREAL; // Initial output value. Restored on Reset.
	_fRate       : LREAL; // Rate of change in units per second. Negative values produce a falling ramp.
END_VAR

METHOD FB_init : BOOL
VAR_INPUT
	bInitRetains : BOOL;  // if TRUE, the retain variables are initialized (warm start / cold start)
	bInCopyCode  : BOOL;  // if TRUE, the instance afterwards gets moved into the copy code (online change)
	fStartValue  : LREAL; // Initial output value.
	fRate        : LREAL; // Rate of change in units per second. Negative values produce a falling ramp.
END_VAR
THIS^._fStartValue := fStartValue;
THIS^._fRate       := fRate;
END_METHOD

(*
Gets or sets the rate of change in units per second.

A positive value produces a rising ramp, a negative value a falling ramp.
Changes take effect immediately.
*)
PROPERTY Rate : LREAL
GET
Rate := THIS^._fRate;
END_GET
SET
THIS^._fRate := Rate;
END_SET
END_PROPERTY

(* Resets the output to the start value set in ``FB_init``. The rate is unaffected. *)
METHOD Reset
VAR_INPUT
END_VAR
THIS^._fOutput := THIS^._fStartValue;
END_METHOD

(*
Advances the ramp by one time step.

.. note::
   Must be called once per cycle on a single PLC task. If the measured cycle
   time is zero the method returns early without updating the output.
*)
METHOD Run
VAR_INST
	{attribute 'hide'}
	bInit : BOOL := TRUE;
	{attribute 'hide'}
	fT    : LREAL;
	{attribute 'hide'}
	fbTaskCycle : FsCommon.FB_PlcTaskCycleChangeDetector(0);
END_VAR
IF bInit THEN
	fT := TO_LREAL(FsCommon.F_GetCurrentTaskCycleTime()) / TO_LREAL(LTIME#1S);
	RETURN(bInit := fT <= 0);
	fbTaskCycle.TaskIndex := FsCommon.F_GetCurrentTaskIndex();
END_IF

RETURN(NOT fbTaskCycle.HasChanged);

THIS^._fOutput := THIS^._fOutput + THIS^._fRate * fT;
END_METHOD

(*
Gets or sets the start value.

This is the output value the ramp returns to after a :meth:`Reset`.
*)
PROPERTY StartValue  : LREAL
GET
StartValue := THIS^._fStartValue;
END_GET
SET
THIS^._fStartValue := StartValue;
END_SET
END_PROPERTY

END_FUNCTION_BLOCK

// Signals/FB_SawtoothWave
(*
Generates a sawtooth wave signal.

The output rises linearly from ``-Amplitude`` to ``+Amplitude`` over one full
cycle then resets instantly, or falls from ``+Amplitude`` to ``-Amplitude``
depending on :attr:`Direction`. :attr:`Bias` shifts the output vertically.

:attr:`Phase` shifts the wave horizontally in radians. Negative values shift
in the opposite direction.

.. note::
   The block is ``FINAL`` and must be instantiated, not extended.
   Use ``FB_init`` to set :attr:`tPeriod`, :attr:`fAmplitude`, :attr:`fBias` and
   :attr:`fPhase` at declaration time.
*)
{attribute 'enable_dynamic_creation'}
{attribute 'no_explicit_call' := 'direct call for this function block is not allowed'}
FUNCTION_BLOCK FINAL FB_SawtoothWave EXTENDS FB_PeriodicSignal
IMPLEMENTS FsCommon.I_Runnable, I_Resettable
VAR
	_eDirection : E_RampDirection; // Direction of the sawtooth. Rising goes from -Amplitude to +Amplitude, Falling goes from +Amplitude to -Amplitude.
	{attribute 'hide'}
	_tTime      : LTIME;
END_VAR

(*
Gets or sets the direction of the sawtooth.

:attr:`~E_RampDirection.Rising` ramps from ``-Amplitude`` to ``+Amplitude``
before resetting. :attr:`~E_RampDirection.Falling` is the inverse.
Changes take effect immediately.
*)
PROPERTY Direction : E_RampDirection
GET
Direction := THIS^._eDirection;
END_GET
SET
THIS^._eDirection := Direction;
END_SET
END_PROPERTY

METHOD FB_init : BOOL
VAR_INPUT
	bInitRetains : BOOL; // if TRUE, the retain variables are initialized (warm start / cold start)
	bInCopyCode : BOOL;  // if TRUE, the instance afterwards gets moved into the copy code (online change)
	tPeriod      : LTIME; // Duration of one full cycle.
	fAmplitude   : LREAL; // Scales the wave. Output swings between Bias ± Amplitude.
	fBias        : LREAL; // Shifts the output vertically.
	fPhase       : LREAL; // Phase offset in radians. Shifts the wave horizontally.
END_VAR
THIS^._tPeriod    := tPeriod;
THIS^._fAmplitude := fAmplitude;
THIS^._fBias      := fBias;
THIS^._fPhase     := fPhase;
END_METHOD

(* Restarts the wave from the beginning by resetting the accumulated time to zero. The phase, amplitude, and bias are unaffected. *)
METHOD Reset
VAR_INPUT
END_VAR
THIS^._tTime := LTIME#0S;
END_METHOD

(*
Advances the sawtooth wave by one time step.

.. note::
   Must be called once per cycle on a single PLC task. If the measured cycle
   time is zero or :attr:`Period` is zero, the method returns early without
   updating the output.
*)
METHOD Run
VAR_INST
	{attribute 'hide'}
	bInit       : BOOL := TRUE;
	{attribute 'hide'}
	fT          : LREAL;
	{attribute 'hide'}
	fbTaskCycle : FsCommon.FB_PlcTaskCycleChangeDetector(0);
END_VAR
VAR
	fPeriod     : LREAL;
	fPhaseTime  : LREAL;
	fCyclePos   : LREAL;
END_VAR
IF bInit THEN
	fT := TO_LREAL(FsCommon.F_GetCurrentTaskCycleTime()) / TO_LREAL(LTIME#1S);
	RETURN(bInit := fT <= 0);
	fbTaskCycle.TaskIndex := FsCommon.F_GetCurrentTaskIndex();
END_IF

RETURN(THIS^._tPeriod <= LTIME#0S OR NOT fbTaskCycle.HasChanged);

THIS^._tTime := THIS^._tTime + TO_LTIME(LREAL_TO_ULINT(fT * 1.0E9));

fPeriod    := TO_LREAL(THIS^._tPeriod) / TO_LREAL(LTIME#1S);
fPhaseTime := TO_LREAL(THIS^._tTime) / TO_LREAL(LTIME#1S) + (THIS^._fPhase / (2.0 * Tc2_System.PI)) * fPeriod;
fCyclePos  := Tc2_Math.LMOD(fPhaseTime, fPeriod) / fPeriod;

CASE THIS^._eDirection OF
	E_RampDirection.Rising:
		THIS^._fOutput := THIS^._fAmplitude * (2.0 * fCyclePos - 1.0) + THIS^._fBias;
	E_RampDirection.Falling:
		THIS^._fOutput := THIS^._fAmplitude * (1.0 - 2.0 * fCyclePos) + THIS^._fBias;
END_CASE
END_METHOD

END_FUNCTION_BLOCK

// Signals/FB_SineWave
(*
Generates a sine wave signal.

The output follows:

.. math::

   y(t) = A \sin\left(\frac{2\pi}{T} t + \phi\right) + B

where :math:`A` is :attr:`Amplitude`, :math:`T` is :attr:`Period` in seconds,
:math:`\phi` is :attr:`Phase` in radians, and :math:`B` is :attr:`Bias`.

.. note::
   The block is ``FINAL`` and must be instantiated, not extended.
   Use ``FB_init`` to set :attr:`tPeriod`, :attr:`fAmplitude`, :attr:`fBias`,
   and :attr:`fPhase` at declaration time.
*)
{attribute 'enable_dynamic_creation'}
{attribute 'no_explicit_call' := 'direct call for this function block is not allowed'}
FUNCTION_BLOCK FINAL FB_SineWave EXTENDS FB_PeriodicSignal
IMPLEMENTS FsCommon.I_Runnable, I_Resettable
VAR
	{attribute 'hide'}
	_tTime : LTIME;
END_VAR

METHOD FB_init : BOOL
VAR_INPUT
	bInitRetains : BOOL; // if TRUE, the retain variables are initialized (warm start / cold start)
	bInCopyCode : BOOL;  // if TRUE, the instance afterwards gets moved into the copy code (online change)
	tPeriod      : LTIME; // Duration of one full cycle.
	fAmplitude   : LREAL; // Scales the wave. Output swings between Bias ± Amplitude.
	fBias        : LREAL; // Shifts the output vertically.
	fPhase       : LREAL; // Phase offset in radians. Shifts the wave horizontally.
END_VAR
THIS^._tPeriod    := tPeriod;
THIS^._fAmplitude := fAmplitude;
THIS^._fBias      := fBias;
THIS^._fPhase     := fPhase;
END_METHOD

(* Restarts the wave from the beginning by resetting the accumulated time to zero. The phase, amplitude, and bias are unaffected. *)
METHOD Reset
VAR_INPUT
END_VAR
THIS^._tTime := LTIME#0S;
END_METHOD

(*
Advances the sine wave by one time step.

.. note::
   Must be called once per cycle on a single PLC task. If the measured cycle
   time is zero or :attr:`Period` is zero, the method returns early without
   updating the output.
*)
METHOD Run
VAR_INST
	{attribute 'hide'}
	bInit       : BOOL := TRUE;
	{attribute 'hide'}
	fT          : LREAL;
	{attribute 'hide'}
	fbTaskCycle : FsCommon.FB_PlcTaskCycleChangeDetector(0);
END_VAR
VAR
	fPeriod : LREAL;
END_VAR
IF bInit THEN
	fT := TO_LREAL(FsCommon.F_GetCurrentTaskCycleTime()) / TO_LREAL(LTIME#1S);
	RETURN(bInit := fT <= 0);
	fbTaskCycle.TaskIndex := FsCommon.F_GetCurrentTaskIndex();
END_IF

RETURN(THIS^._tPeriod <= LTIME#0S OR NOT fbTaskCycle.HasChanged);

THIS^._tTime := THIS^._tTime + TO_LTIME(LREAL_TO_ULINT(fT * 1.0E9));

fPeriod := TO_LREAL(THIS^._tPeriod) / TO_LREAL(LTIME#1S);

THIS^._fOutput := THIS^._fAmplitude 
	* SIN((2.0 * Tc2_System.PI / fPeriod) * (TO_LREAL(THIS^._tTime) / TO_LREAL(LTIME#1S)) + THIS^._fPhase) 
	+ THIS^._fBias;
END_METHOD

END_FUNCTION_BLOCK

// Signals/FB_SquareWave
(*
Generates a square wave signal.

The raw wave alternates between ``+1`` and ``-1`` over one period. :attr:`Amplitude`
scales the wave and :attr:`Bias` shifts it vertically, giving an output that swings
between ``Bias + Amplitude`` and ``Bias - Amplitude``.

:attr:`Phase` shifts the wave horizontally in radians. A phase of π starts the
wave in its low half-cycle, a phase of -π has the same effect.

.. note::
   The block is ``FINAL`` and must be instantiated, not extended.
   Use ``FB_init`` to set :attr:`tPeriod`, :attr:`fAmplitude`, :attr:`fBias`,
   and :attr:`fPhase` at declaration time.
*)
{attribute 'enable_dynamic_creation'}
{attribute 'no_explicit_call' := 'direct call for this function block is not allowed'}
FUNCTION_BLOCK FINAL FB_SquareWave EXTENDS FB_PeriodicSignal
IMPLEMENTS FsCommon.I_Runnable, I_Resettable
VAR
	{attribute 'hide'}
	_tTime : LTIME; // Accumulated time.
END_VAR

METHOD FB_init : BOOL
VAR_INPUT
	bInitRetains : BOOL;  // if TRUE, the retain variables are initialized (warm start / cold start)
	bInCopyCode  : BOOL;  // if TRUE, the instance afterwards gets moved into the copy code (online change)
	tPeriod      : LTIME; // Duration of one full cycle.
	fAmplitude   : LREAL; // Scales the ±1 wave. Output swings between Bias ± Amplitude.
	fBias        : LREAL; // Shifts the output up or down by a fixed value.
	fPhase       : LREAL; // Phase offset in radians. Shifts the wave horizontally. Negative values shift in the opposite direction.
END_VAR
THIS^._tPeriod    := tPeriod;
THIS^._fAmplitude := fAmplitude;
THIS^._fBias      := fBias;
THIS^._fPhase     := fPhase;
END_METHOD

(* Restarts the wave from the beginning by resetting the accumulated time to zero. The phase, amplitude, and bias are unaffected. *)
METHOD Reset
VAR_INPUT
END_VAR
THIS^._tTime := LTIME#0S;
END_METHOD

(*
Advances the square wave by one time step.

.. note::
   Must be called once per cycle on a single PLC task. If the measured cycle
   time is zero or :attr:`Period` is zero, the method returns early without
   updating the output.
*)
METHOD Run
VAR_INST
	{attribute 'hide'}
	bInit 		 : BOOL := TRUE;
	{attribute 'hide'}
	tT           : LTIME;
	{attribute 'hide'}
	fbTaskCycle  :  FsCommon.FB_PlcTaskCycleChangeDetector(0);
END_VAR
VAR
	fCyclePhase  : LREAL;
	fPeriod		 : LREAL;
END_VAR
IF bInit THEN
	tT := FsCommon.F_GetCurrentTaskCycleTime();
	RETURN(bInit := tT = LTIME#0S);
	fbTaskCycle.TaskIndex := FsCommon.F_GetCurrentTaskIndex();
END_IF

RETURN(THIS^._tPeriod <= LTIME#0S OR NOT fbTaskCycle.HasChanged);

THIS^._tTime := THIS^._tTime + tT;

fPeriod := TO_LREAL(THIS^._tPeriod) / TO_LREAL(LTIME#1S);

fCyclePhase := Tc2_Math.LMOD(
	(TO_LREAL(THIS^._tTime) / TO_LREAL(LTIME#1S)) + ((THIS^._fPhase / (2.0 * Tc2_System.PI)) * fPeriod), 
	fPeriod
) / fPeriod;

IF fCyclePhase < 0.5 THEN
	THIS^._fOutput :=  THIS^._fAmplitude + THIS^._fBias;
ELSE
	THIS^._fOutput := -THIS^._fAmplitude + THIS^._fBias;
END_IF
END_METHOD

END_FUNCTION_BLOCK

// Signals/FB_TriangleWave
(*
Generates a triangle wave signal.

The output rises linearly from ``-Amplitude`` to ``+Amplitude`` over the first
half-cycle, then falls back to ``-Amplitude`` over the second half. :attr:`Bias`
shifts the output vertically.

:attr:`Phase` shifts the wave horizontally in radians. A phase of π starts the
wave at its peak rather than its trough.

.. note::
   The block is ``FINAL`` and must be instantiated, not extended.
   Use ``FB_init`` to set :attr:`tPeriod`, :attr:`fAmplitude`, :attr:`fBias`,
   and :attr:`fPhase` at declaration time.
*)
{attribute 'enable_dynamic_creation'}
{attribute 'no_explicit_call' := 'direct call for this function block is not allowed'}
FUNCTION_BLOCK FINAL FB_TriangleWave EXTENDS FB_PeriodicSignal
IMPLEMENTS FsCommon.I_Runnable, I_Resettable
VAR
	{attribute 'hide'}
	_tTime : LTIME;
END_VAR

METHOD FB_init : BOOL
VAR_INPUT
	bInitRetains : BOOL; // if TRUE, the retain variables are initialized (warm start / cold start)
	bInCopyCode : BOOL;  // if TRUE, the instance afterwards gets moved into the copy code (online change)
	tPeriod      : LTIME; // Duration of one full cycle.
	fAmplitude   : LREAL; // Scales the wave. Output swings between Bias ± Amplitude.
	fBias        : LREAL; // Shifts the output vertically.
	fPhase       : LREAL; // Phase offset in radians. Shifts the wave horizontally.
END_VAR
THIS^._tPeriod    := tPeriod;
THIS^._fAmplitude := fAmplitude;
THIS^._fBias      := fBias;
THIS^._fPhase     := fPhase;
END_METHOD

(* Restarts the wave from the beginning by resetting the accumulated time to zero. The phase, amplitude, and bias are unaffected. *)
METHOD Reset
VAR_INPUT
END_VAR
THIS^._tTime := LTIME#0S;
END_METHOD

(*
Advances the triangle wave by one time step.

.. note::
   Must be called once per cycle on a single PLC task. If the measured cycle
   time is zero or :attr:`Period` is zero, the method returns early without
   updating the output.
*)
METHOD Run
VAR_INST
	{attribute 'hide'}
	bInit       : BOOL := TRUE;
	{attribute 'hide'}
	fT          : LREAL;
	{attribute 'hide'}
	fbTaskCycle : FsCommon.FB_PlcTaskCycleChangeDetector(0);
END_VAR
VAR
	fPeriod     : LREAL;
	fPhaseTime  : LREAL;
	fCyclePos   : LREAL;
END_VAR
IF bInit THEN
	fT := TO_LREAL(FsCommon.F_GetCurrentTaskCycleTime()) / TO_LREAL(LTIME#1S);
	RETURN(bInit := fT <= 0);
	fbTaskCycle.TaskIndex := FsCommon.F_GetCurrentTaskIndex();
END_IF

RETURN(THIS^._tPeriod <= LTIME#0S OR NOT fbTaskCycle.HasChanged);

THIS^._tTime := THIS^._tTime + TO_LTIME(LREAL_TO_ULINT(fT * 1.0E9));

fPeriod    := TO_LREAL(THIS^._tPeriod) / TO_LREAL(LTIME#1S);
fPhaseTime := TO_LREAL(THIS^._tTime) / TO_LREAL(LTIME#1S) + (THIS^._fPhase / (2.0 * Tc2_system.PI)) * fPeriod;
fCyclePos  := Tc2_Math.LMOD(fPhaseTime, fPeriod) / fPeriod;

IF fCyclePos < 0.5 THEN
	THIS^._fOutput := THIS^._fAmplitude * (4.0 * fCyclePos - 1.0) + THIS^._fBias;
ELSE
	THIS^._fOutput := THIS^._fAmplitude * (3.0 - 4.0 * fCyclePos) + THIS^._fBias;
END_IF
END_METHOD

END_FUNCTION_BLOCK

// Simulation/FB_SecondOrderPlant
(*
Simulates a second-order linear plant using the Tustin (bilinear) discretisation
with frequency pre-warping to preserve the natural frequency :attr:`Wn` exactly.

The continuous-time transfer function is:

.. math::

   G(s) = \frac{K \omega_n^2}{s^2 + 2 \zeta \omega_n s + \omega_n^2}

where :math:`K` is :attr:`Gain`, :math:`\omega_n` is :attr:`Wn`, and
:math:`\zeta` is :attr:`Zeta`.

.. note::
   The block is ``FINAL`` and must be instantiated, not extended.
   Use ``FB_init`` to set :attr:`fGain`, :attr:`fWn`, and :attr:`fZeta` at declaration time.
*)
{attribute 'enable_dynamic_creation'}
{attribute 'no_explicit_call' := 'direct call for this function block is not allowed'}
FUNCTION_BLOCK FINAL FB_SecondOrderPlant EXTENDS FB_SisoComponent
IMPLEMENTS FsCommon.I_Runnable, I_Resettable
VAR
	_fGain 	: LREAL; // Steady-state gain (K). Ratio of output to input once the plant has fully settled.
	_fWn 	: LREAL; // Natural frequency, rad/s), sets how fast the plant responds.
	_fZeta	: LREAL; // Damping ratio. Less than 1 gives overshoot, 1 is critically damped, greater than 1 is overdamped.
	{attribute 'hide'}
	_fY1    : LREAL; // y[k-1]
	{attribute 'hide'}
    _fY2    : LREAL; // y[k-2]
	{attribute 'hide'}
    _fU1    : LREAL; // u[k-1]
	{attribute 'hide'}
    _fU2    : LREAL; // u[k-2]
END_VAR

METHOD FB_init : BOOL
VAR_INPUT
	bInitRetains : BOOL;  // if TRUE, the retain variables are initialized (warm start / cold start)
	bInCopyCode  : BOOL;  // if TRUE, the instance afterwards gets moved into the copy code (online change)
	fGain 		 : LREAL; // Steady-state gain (K). Ratio of output to input once the plant has fully settled.
	fWn 		 : LREAL; // Natural frequency in rad/s. Controls how fast the plant responds.
	fZeta 		 : LREAL; // Damping ratio. Less than 1 gives overshoot, 1 is critically damped, greater than 1 is overdamped.
END_VAR
THIS^._fGain := fGain;
THIS^._fWn 	 := fWn;
THIS^._fZeta := fZeta;
END_METHOD

(*
Gets or sets the steady-state gain.

This is the factor by which a constant input is scaled to produce the output once
the plant has fully settled. For example, a gain of 2 with a constant input of 5
will eventually produce an output of 10.
*)
PROPERTY Gain : LREAL
GET
Gain := THIS^._fGain;
END_GET
SET
THIS^._fGain := Gain;
END_SET
END_PROPERTY

(* Sets the output and all internal state to zero, returning the plant to its initial conditions. *)
METHOD Reset
VAR_INPUT
END_VAR
THIS^._fOutput := 0;
THIS^._fY1     := 0;
THIS^._fY2     := 0;
THIS^._fU1     := 0;
THIS^._fU2     := 0;
END_METHOD

(*
Advances the plant by one time step.

.. note::
   Must be called once per cycle on a single PLC task. This is because on the 
   first call, the cycle time is measured and stored for use in all subsequent calls. 
 
   If the cycle time is zero or :attr:`Wn` is zero, the method returns early 
   without updating the output.
*)
METHOD Run
VAR_INST
	{attribute 'hide'}
	bInit 		 	: BOOL := TRUE;
	{attribute 'hide'}
	fT				 	: LREAL;
	{attribute 'hide'}
	fbTaskCycle 		:  FsCommon.FB_PlcTaskCycleChangeDetector(0);
END_VAR
VAR
	fWd, fWd2, fT2, fDen  : LREAL;
    fA1, fA2         : LREAL;
    fB0, fB1, fB2    : LREAL;
    fY               : LREAL;
END_VAR
IF bInit THEN
	fT := TO_LREAL(FsCommon.F_GetCurrentTaskCycleTime()) / TO_LREAL(LTIME#1S);
	RETURN(bInit := fT <= 0);
	fbTaskCycle.TaskIndex := FsCommon.F_GetCurrentTaskIndex();
	END_IF

RETURN(THIS^._fWn <= 0 OR NOT fbTaskCycle.HasChanged);

// Pre-warp natural frequency to preserve Wn exactly under Tustin
fWd  := (2.0 / fT) * TAN(THIS^._fWn * fT / 2.0);
fWd2 := fWd * fWd;
fT2  := fT * fT;
fDen := (4.0 / fT2) + 2.0 * THIS^._fZeta * fWd * (2.0 / fT) + fWd2;

fB0 := (THIS^._fGain * fWd2) / fDen;
fB1 := (2.0 * THIS^._fGain * fWd2) / fDen;
fB2 := fB0;

fA1 := ((-8.0 / fT2) + 2.0 * fWd2) / fDen;
fA2 := ((4.0 / fT2) - 2.0 * THIS^._fZeta * fWd * (2.0 / fT) + fWd2) / fDen;

fY := fB0 * THIS^._fInput + fB1 * THIS^._fU1 + fB2 * THIS^._fU2
       - fA1 * THIS^._fOutput - fA2 * THIS^._fY1;

THIS^._fY2      := THIS^._fY1;
THIS^._fY1      := THIS^._fOutput;
THIS^._fU2      := THIS^._fU1;
THIS^._fU1      := THIS^._fInput;
THIS^._fOutput 	:= fY;
END_METHOD

(*
Gets or sets the natural frequency in rad/s.

This controls the speed of the plant's response. 
A higher value means a faster response. To convert from Hz, multiply by 2π.
*)
PROPERTY Wn : LREAL
GET
Wn := THIS^._fWn;
END_GET
SET
THIS^._fWn := Wn;
END_SET
END_PROPERTY

(* 
Gets or sets the damping ratio.

This controls the shape of the response.
  - A value below 1 produces an oscillating response that overshoots before settling. 
  - A value of exactly 1 (critically damped) settles as fast as possible without any overshoot.
  - A value above 1 settles more slowly with no overshoot.
*)
PROPERTY Zeta : LREAL
GET
Zeta := THIS^._fZeta;
END_GET
SET
THIS^._fZeta := Zeta;
END_SET
END_PROPERTY

END_FUNCTION_BLOCK
